// TIA Portal V20 export
TYPE "UDT_PartState"
   STRUCT
      Good : Bool;
      Unknown : Bool;
      Bad : Bool;
      Absent : Bool;
      PresentUnexpected : Bool;
      AbsentUnexpected : Bool;
   END_STRUCT;
END_TYPE
